FUNCTION_BLOCK FB_Component EXTENDS FB_BaseComponent IMPLEMENTS ITF_Component, ITF_Component_HMI_Init
VAR
	
END_VAR

(*			
	EVERDE sp. z o.o.
	Rafał Osajda		24.03.2025		TC 4024.66
	Definicja nowego zgłoszenia
*)
METHOD PUBLIC EventsDefinition : BOOL
VAR_INPUT
END_VAR

VAR
	stName: ST_Label;
END_VAR
SUPER^.EventsDefinition ();

THIS^.AddEvent (
	bIgnorujPowtorzenia		:= TRUE,
	eRodzajZdarzenia		:= E_BaseEvents_Type.ALARM,
	bWymagaZatwierdzenia	:=FALSE,
	stOpis					:= stName
);
END_METHOD

END_FUNCTION_BLOCK

(* stored: Version 1.1.0.1, ProductVersion 3.1.4024.15
   POU FB_Component: Id {2de1b166-2e29-435f-8ec0-de550667ad0a}, SpecialFunc None
   Folder Events: Id {7bb4e45e-1048-4dff-a472-983f58eabfc3}
   Method EventsDefinition: Id {a55dd4c8-65f3-4ae1-b770-b8a090b813df} *)
